FUNCTION_BLOCK PUBLIC TmsExchange EXTENDS Process
VAR_INPUT
	TmsSwitch : ITF_TmsSwitch;
	StateMachine : IPmlStateMachine;
END_VAR
VAR_OUTPUT
END_VAR
VAR
	holdingStation : TmsHoldStation;
	embarkingStation : TmsEmbarkStation;
END_VAR

holdingStation(StateMachine := StateMachine, embarkStation := embarkingStation);
embarkingStation(StateMachine := StateMachine, TmsSwitch := TmsSwitch);

PROPERTY EmbarkStation : IProcess
GET
EmbarkStation := embarkingStation;
END_GET
END_PROPERTY

PROPERTY ExchangeTrackLevel : int
GET
ExchangeTrackLevel := embarkingStation.TrackLevel;
END_GET
SET
embarkingStation.TrackLevel := ExchangeTrackLevel;
END_SET
END_PROPERTY

PROPERTY HoldStation : IProcess
GET
HoldStation := holdingStation;
END_GET
END_PROPERTY

PROPERTY SwitchTravelPosition : MC_LREAL
GET
SwitchTravelPosition := embarkingStation.SwitchTravelPosition;
END_GET
SET
embarkingStation.SwitchTravelPosition := SwitchTravelPosition;
END_SET
END_PROPERTY

END_FUNCTION_BLOCK

(* stored: Version 1.1.0.1, ProductVersion 3.1.4024.12
   POU TmsExchange: Id {27fb18f6-f27b-4462-bf40-a5ac4ef58917}, SpecialFunc None
   Property EmbarkStation: Id {ad3c6c49-301b-4ffc-ba92-cb113791b6b6}
   Get Get: Id {affd081c-0ef5-41a6-95e9-3ca51e2a37b1}
   Property ExchangeTrackLevel: Id {a9874efe-b6f7-44a3-97fb-b9da1b2bb67f}
   Get Get: Id {b227262b-022a-4f6f-949f-c433e85e026a}
   Set Set: Id {1749dfec-ed0e-4ade-93c1-5b9f22c6671c}
   Property HoldStation: Id {fd38c671-f96a-44ac-a7b5-6af55bf1cbe4}
   Get Get: Id {4becc177-9df4-4fa7-ab85-81067137af39}
   Property SwitchTravelPosition: Id {1475f196-d2b7-4273-b2f6-2690b7930f9c}
   Get Get: Id {6209c32e-023d-4b82-9ce1-001f86156112}
   Set Set: Id {55de1914-4dbc-4c4e-8277-42747693dd1e} *)
